// TIA Portal project "13_Buffer_Station" (V19)

(* hardware
DEVICE "S7-1500/ET200MP station_1"  S7-1500 station
   slot 0: "Rail_0"  Rack  6ES7 590-1***0-0AA0
   slot 1: "PLC_1"  CPU 1513-1 PN  6ES7 513-1AL02-0AB0  V2.9
      slot 3: "CPU display_1"  6ES7591-1AA00-0AA0
      slot 32768: "PROFINET interface_1"  X1
         slot 32769: "Port_1"  X1 P1
         slot 32770: "Port_2"  X1 P2
      slot 34817: "Virtual CP interface port_1"  Virtual CP interface port  Virtual CP interface port
*)

// ===== PLC "PLC_1"  CPU 1513-1 PN =====

VAR_GLOBAL   // PLC tag table "Default tag table"
   "nw2" AT %M0.0 : Bool;
   "nw3 2nd memory (Pause)" AT %M0.2 : Bool;
   "nw3 1st memory (Unpause)" AT %M0.1 : Bool;
   "nw3 return" AT %M4.0 : Bool;
   "nw4" AT %M0.3 : Bool;
   "nw6 ae p" AT %M1.3 : Bool;
   "nw6 1st SR" AT %M0.5 : Bool;
   "nw6 abe p" AT %M0.7 : Bool;
   "nw6 abe p2" AT %M1.4 : Bool;
   "nw6 2nd SR" AT %M1.5 : Bool;
   "nw6 ae p2" AT %M1.6 : Bool;
   "nw5" AT %M0.4 : Bool;
   "nw7 1st SR" AT %M0.6 : Bool;
   "I/P for exit conveyor" AT %MD100 : Real;
   "nw7 2nd SR" AT %M1.7 : Bool;
   "nw8 abe p" AT %M1.1 : Bool;
   "nw8" AT %M1.0 : Bool;
   "nw8 ae p" AT %M1.2 : Bool;
   "nw8 ret" AT %M2.0 : Bool;
   "Convert potention meter value from Real to DINT" AT %MD110 : Real;
   "Store MD110 here & send to QD42" AT %MD10 : DInt;
   "nw9 ae p1" AT %M2.2 : Bool;
   "nw9 1st SR" AT %M2.1 : Bool;
   "nw9 abe p1" AT %M2.3 : Bool;
   "nw9 abe p2" AT %M2.4 : Bool;
   "nw9 ae p2" AT %M2.5 : Bool;
   "nw9 abe p3" AT %M2.7 : Bool;
   "nw9 2nd SR" AT %M2.6 : Bool;
   "nw9 ae p3" AT %M3.0 : Bool;
   "nw10 1st SR" AT %M3.1 : Bool;
   "I/P for exit conveyor (set)" AT %MD120 : Real;
   "nw10 2nd SR" AT %M3.2 : Bool;
   "nw11 abe p1" AT %M3.4 : Bool;
   "nw11" AT %M3.3 : Bool;
   "nw11 ae p1" AT %M3.6 : Bool;
   "nw11 ae p2" AT %M3.5 : Bool;
   "nw11 abe p2" AT %M3.7 : Bool;
END_VAR

VAR_GLOBAL   // PLC tag table "Tag table from XML_1"
   "Start" AT %I0.0 : Bool;
   "Pause & Unpause" AT %I0.1 : Bool;
   "Reset" AT %I0.2 : Bool;
   "At buffer entry" AT %I0.3 : Bool;
   "At buffer exit" AT %I0.4 : Bool;
   "At exit" AT %I0.5 : Bool;
   "Without set (mode)" AT %I0.6 : Bool;
   "Send set (mode)" AT %I0.7 : Bool;
   "Start light" AT %Q0.0 : Bool;
   "P & UP light" AT %Q0.1 : Bool;
   "Reset light" AT %Q0.2 : Bool;
   "Stop blade" AT %Q0.3 : Bool;
   "Buffer Vel." AT %ID30 : Real;
   "Set the value for boxes" AT %ID34 : Real;
   "Buffer conveyor" AT %QD30 : Real;
   "Exit conveyor" AT %QD34 : Real;
   "Display Buffer (Speed)" AT %QD38 : Real;
   "Display for set of boxes" AT %QD42 : DInt;
   "Display Counter" AT %QD46 : DInt;
END_VAR

// folder: System blocks/Program resources

DATA_BLOCK "IEC_Counter_0_DB"   // DB1
{ S7_Optimized_Access := 'TRUE' }
AUTHOR : Simatic
FAMILY : IEC
NAME : CNTR
VERSION : 1.0
// stored: InstanceOfName IEC_COUNTER
"IEC_COUNTER"
BEGIN
END_DATA_BLOCK

DATA_BLOCK "IEC_Counter_0_DB_1"   // DB2
{ S7_Optimized_Access := 'TRUE' }
AUTHOR : SIMATIC
FAMILY : IEC
NAME : DCNTR
VERSION : 1.2
// stored: InstanceOfName IEC_DCOUNTER
"IEC_DCOUNTER"
BEGIN
END_DATA_BLOCK

DATA_BLOCK "IEC_Counter_0_DB_2"   // DB3
{ S7_Optimized_Access := 'TRUE' }
AUTHOR : SIMATIC
FAMILY : IEC
NAME : DCNTR
VERSION : 1.2
// stored: InstanceOfName IEC_DCOUNTER
"IEC_DCOUNTER"
BEGIN
END_DATA_BLOCK

DATA_BLOCK "IEC_Counter_0_DB_3"   // DB4
{ S7_Optimized_Access := 'TRUE' }
AUTHOR : SIMATIC
FAMILY : IEC
NAME : DCNTR
VERSION : 1.2
// stored: InstanceOfName IEC_DCOUNTER
"IEC_DCOUNTER"
BEGIN
END_DATA_BLOCK

DATA_BLOCK "IEC_Counter_0_DB_4"   // DB5
{ S7_Optimized_Access := 'TRUE' }
AUTHOR : SIMATIC
FAMILY : IEC
NAME : DCNTR
VERSION : 1.2
// stored: InstanceOfName IEC_DCOUNTER
"IEC_DCOUNTER"
BEGIN
END_DATA_BLOCK

// folder: (top level)

ORGANIZATION_BLOCK "Main"   // OB1, LAD, ProgramCycle
TITLE = "Main Program Sweep (Cycle)"
{ S7_Optimized_Access := 'TRUE' }
VERSION : 0.1
   VAR_INPUT
      Initial_Call : Bool;   // Initial call of this OB
      Remanence : Bool;   // =True, if remanent data are available
   END_VAR
   VAR_TEMP   // added for the SCL form of the ladder/FBD networks
      _w1 : Bool;
      _w2 : Bool;
      _w3 : Bool;
      _w4 : Bool;
      _w5 : Bool;
      _w6 : Bool;
   END_VAR
BEGIN

REGION Network 2: Start or Reset System with LED ON/OFF
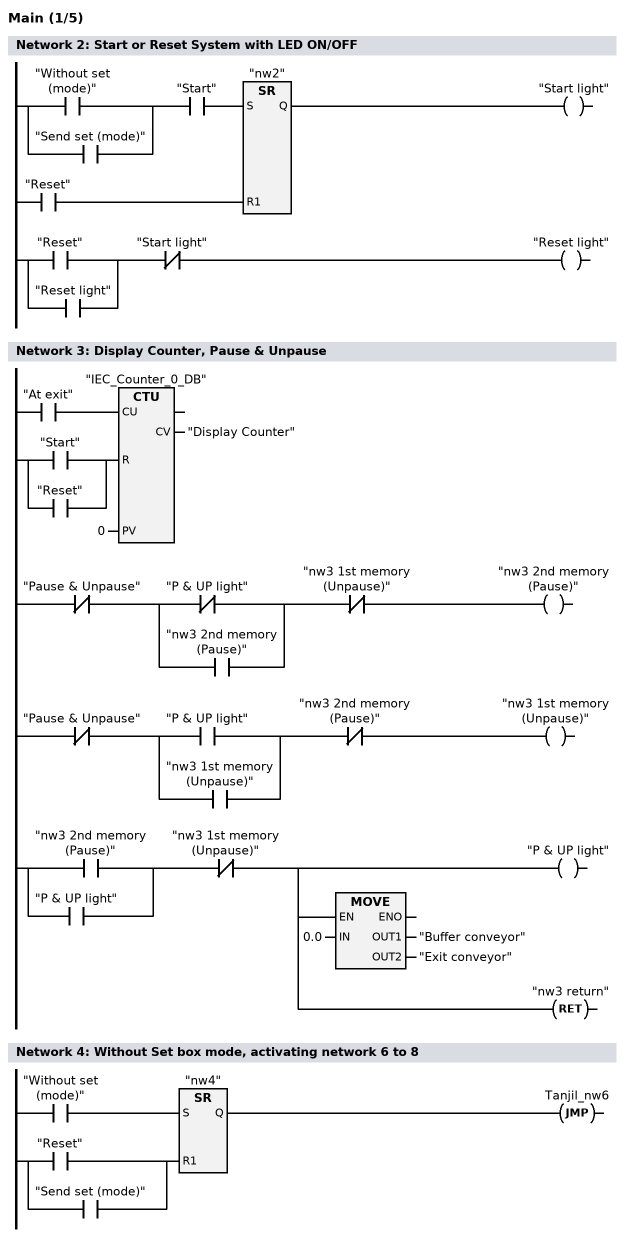
   RUNG wire#powerrail
      Contact( "Without set (mode)" )
      wire#w1
      Contact( "Start" )
      S_SR(operand := "nw2", r1 := wire#w2)
      Coil( "Start light" )
   END_RUNG
   RUNG wire#powerrail
      Contact( "Send set (mode)" )
   END_RUNG wire#w1
   RUNG wire#powerrail
      Contact( "Reset" )
   END_RUNG wire#w2
   RUNG wire#powerrail
      Contact( "Reset" )
      wire#w3
      I_Contact( "Start light" )
      Coil( "Reset light" )
   END_RUNG
   RUNG wire#powerrail
      Contact( "Reset light" )
   END_RUNG wire#w3
   // the same network as SCL:
   IF ("Without set (mode)" OR "Send set (mode)") AND "Start" THEN
       "nw2" := TRUE;   // SR flip-flop
   END_IF;
   IF "Reset" THEN "nw2" := FALSE; END_IF;
   "Start light" := "nw2";
   "Reset light" := ("Reset" OR "Reset light") AND NOT "Start light";
END_REGION

REGION Network 3: Display Counter, Pause & Unpause
   "IEC_Counter_0_DB".CTU(CU := "At exit", R := "Start" OR "Reset", PV := 0, CV => "Display Counter");
   "nw3 2nd memory (Pause)" := NOT "Pause & Unpause" AND (NOT "P & UP light" OR "nw3 2nd memory (Pause)") AND NOT "nw3 1st memory (Unpause)";
   "nw3 1st memory (Unpause)" := NOT "Pause & Unpause" AND ("P & UP light" OR "nw3 1st memory (Unpause)") AND NOT "nw3 2nd memory (Pause)";
   "P & UP light" := ("nw3 2nd memory (Pause)" OR "P & UP light") AND NOT "nw3 1st memory (Unpause)";
   IF "P & UP light" THEN
       "Buffer conveyor" := 0.0;
       "Exit conveyor" := 0.0;
       ENO := "nw3 return";
       RETURN;
   END_IF;
END_REGION

REGION Network 4: Without Set box mode, activating network 6 to 8
   RUNG wire#powerrail
      Contact( "Without set (mode)" )
      S_SR(operand := "nw4", r1 := wire#w1)
      JumpCoil( Tanjil_nw6 )
   END_RUNG
   RUNG wire#powerrail
      Contact( "Reset" )
   END_RUNG wire#w1
   RUNG wire#powerrail
      Contact( "Send set (mode)" )
   END_RUNG wire#w1
   // the same network as SCL:
   IF "Without set (mode)" THEN
       "nw4" := TRUE;   // SR flip-flop
   END_IF;
   IF "Reset" OR "Send set (mode)" THEN "nw4" := FALSE; END_IF;
   IF "nw4" THEN GOTO Tanjil_nw6; END_IF;
END_REGION

REGION Network 5: Activating Network 9 to 11 (sending set of boxes)
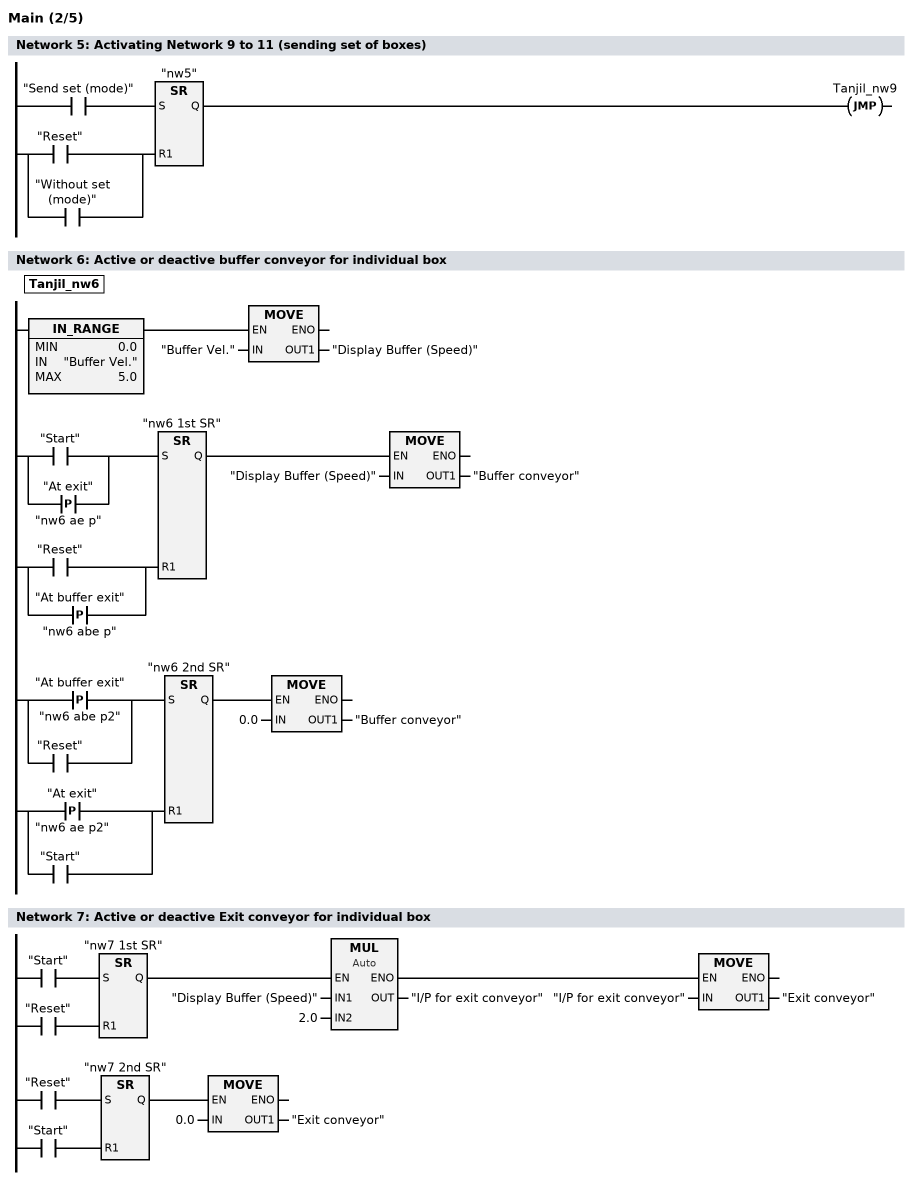
   RUNG wire#powerrail
      Contact( "Send set (mode)" )
      S_SR(operand := "nw5", r1 := wire#w1)
      JumpCoil( Tanjil_nw9 )
   END_RUNG
   RUNG wire#powerrail
      Contact( "Reset" )
   END_RUNG wire#w1
   RUNG wire#powerrail
      Contact( "Without set (mode)" )
   END_RUNG wire#w1
   // the same network as SCL:
   IF "Send set (mode)" THEN
       "nw5" := TRUE;   // SR flip-flop
   END_IF;
   IF "Reset" OR "Without set (mode)" THEN "nw5" := FALSE; END_IF;
   IF "nw5" THEN GOTO Tanjil_nw9; END_IF;
END_REGION

REGION Network 6: Active or deactive buffer conveyor for individual box
   Label( Tanjil_nw6 )
   RUNG wire#powerrail
      { S7_Templates := "SrcType := Real" } InRange(min := 0.0, in := "Buffer Vel.", max := 5.0)
      { S7_GenerateENO := "TRUE" } Move(in := "Buffer Vel.", out1 => "Display Buffer (Speed)")
   END_RUNG
   RUNG wire#powerrail
      Contact( "Start" )
      wire#w1
      S_SR(operand := "nw6 1st SR", r1 := wire#w2)
      { S7_GenerateENO := "TRUE" } Move(in := "Display Buffer (Speed)", out1 => "Buffer conveyor")
   END_RUNG
   RUNG wire#powerrail
      P_Contact(operand := "At exit", bit := "nw6 ae p")
   END_RUNG wire#w1
   RUNG wire#powerrail
      Contact( "Reset" )
   END_RUNG wire#w2
   RUNG wire#powerrail
      P_Contact(operand := "At buffer exit", bit := "nw6 abe p")
   END_RUNG wire#w2
   RUNG wire#powerrail
      P_Contact(operand := "At buffer exit", bit := "nw6 abe p2")
      wire#w3
      S_SR(operand := "nw6 2nd SR", r1 := wire#w4)
      { S7_GenerateENO := "TRUE" } Move(in := 0.0, out1 => "Buffer conveyor")
   END_RUNG
   RUNG wire#powerrail
      Contact( "Reset" )
   END_RUNG wire#w3
   RUNG wire#powerrail
      P_Contact(operand := "At exit", bit := "nw6 ae p2")
   END_RUNG wire#w4
   RUNG wire#powerrail
      Contact( "Start" )
   END_RUNG wire#w4
   // the same network as SCL:
   Tanjil_nw6:
   IF (0.0 <= "Buffer Vel.") AND ("Buffer Vel." <= 5.0) THEN
       "Display Buffer (Speed)" := "Buffer Vel.";
   END_IF;
   #_w1 := "At exit" AND NOT "nw6 ae p";   // rising edge of "At exit"
   "nw6 ae p" := "At exit";
   #_w2 := "At buffer exit" AND NOT "nw6 abe p";   // rising edge of "At buffer exit"
   "nw6 abe p" := "At buffer exit";
   IF "Start" OR #_w1 THEN
       "nw6 1st SR" := TRUE;   // SR flip-flop
   END_IF;
   IF "Reset" OR #_w2 THEN "nw6 1st SR" := FALSE; END_IF;
   IF "nw6 1st SR" THEN "Buffer conveyor" := "Display Buffer (Speed)"; END_IF;
   #_w3 := "At buffer exit" AND NOT "nw6 abe p2";   // rising edge of "At buffer exit"
   "nw6 abe p2" := "At buffer exit";
   #_w4 := "At exit" AND NOT "nw6 ae p2";   // rising edge of "At exit"
   "nw6 ae p2" := "At exit";
   IF #_w3 OR "Reset" THEN
       "nw6 2nd SR" := TRUE;   // SR flip-flop
   END_IF;
   IF #_w4 OR "Start" THEN "nw6 2nd SR" := FALSE; END_IF;
   IF "nw6 2nd SR" THEN "Buffer conveyor" := 0.0; END_IF;
END_REGION

REGION Network 7: Active or deactive Exit conveyor for individual box
   RUNG wire#powerrail
      Contact( "Start" )
      S_SR(operand := "nw7 1st SR", r1 := wire#w1)
      { S7_GenerateENO := "TRUE" } Mul(in1 := "Display Buffer (Speed)", in2 := 2.0, out => "I/P for exit conveyor")
      { S7_GenerateENO := "TRUE" } Move(in := "I/P for exit conveyor", out1 => "Exit conveyor")
   END_RUNG
   RUNG wire#powerrail
      Contact( "Reset" )
   END_RUNG wire#w1
   RUNG wire#powerrail
      Contact( "Reset" )
      S_SR(operand := "nw7 2nd SR", r1 := wire#w2)
      { S7_GenerateENO := "TRUE" } Move(in := 0.0, out1 => "Exit conveyor")
   END_RUNG
   RUNG wire#powerrail
      Contact( "Start" )
   END_RUNG wire#w2
   // the same network as SCL:
   // ENO of a box is taken as its EN; it also drops when the box reports an error
   IF "Start" THEN
       "nw7 1st SR" := TRUE;   // SR flip-flop
   END_IF;
   IF "Reset" THEN "nw7 1st SR" := FALSE; END_IF;
   IF "nw7 1st SR" THEN
       "I/P for exit conveyor" := "Display Buffer (Speed)" * 2.0;
       "Exit conveyor" := "I/P for exit conveyor";
   END_IF;
   IF "Reset" THEN
       "nw7 2nd SR" := TRUE;   // SR flip-flop
   END_IF;
   IF "Start" THEN "nw7 2nd SR" := FALSE; END_IF;
   IF "nw7 2nd SR" THEN "Exit conveyor" := 0.0; END_IF;
END_REGION

REGION Network 8: Active or deactive the STOP Blade
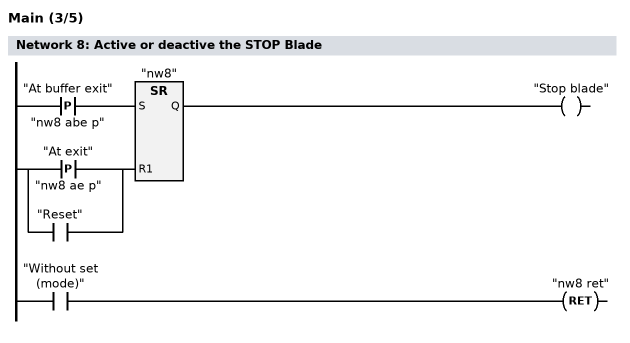
   #_w1 := "At buffer exit" AND NOT "nw8 abe p";   // rising edge of "At buffer exit"
   "nw8 abe p" := "At buffer exit";
   #_w2 := "At exit" AND NOT "nw8 ae p";   // rising edge of "At exit"
   "nw8 ae p" := "At exit";
   IF #_w1 THEN
       "nw8" := TRUE;   // SR flip-flop
   END_IF;
   IF #_w2 OR "Reset" THEN "nw8" := FALSE; END_IF;
   "Stop blade" := "nw8";
   IF "Without set (mode)" THEN
       ENO := "nw8 ret";
       RETURN;
   END_IF;
END_REGION

REGION Network 9: Active Buffer Conveyor
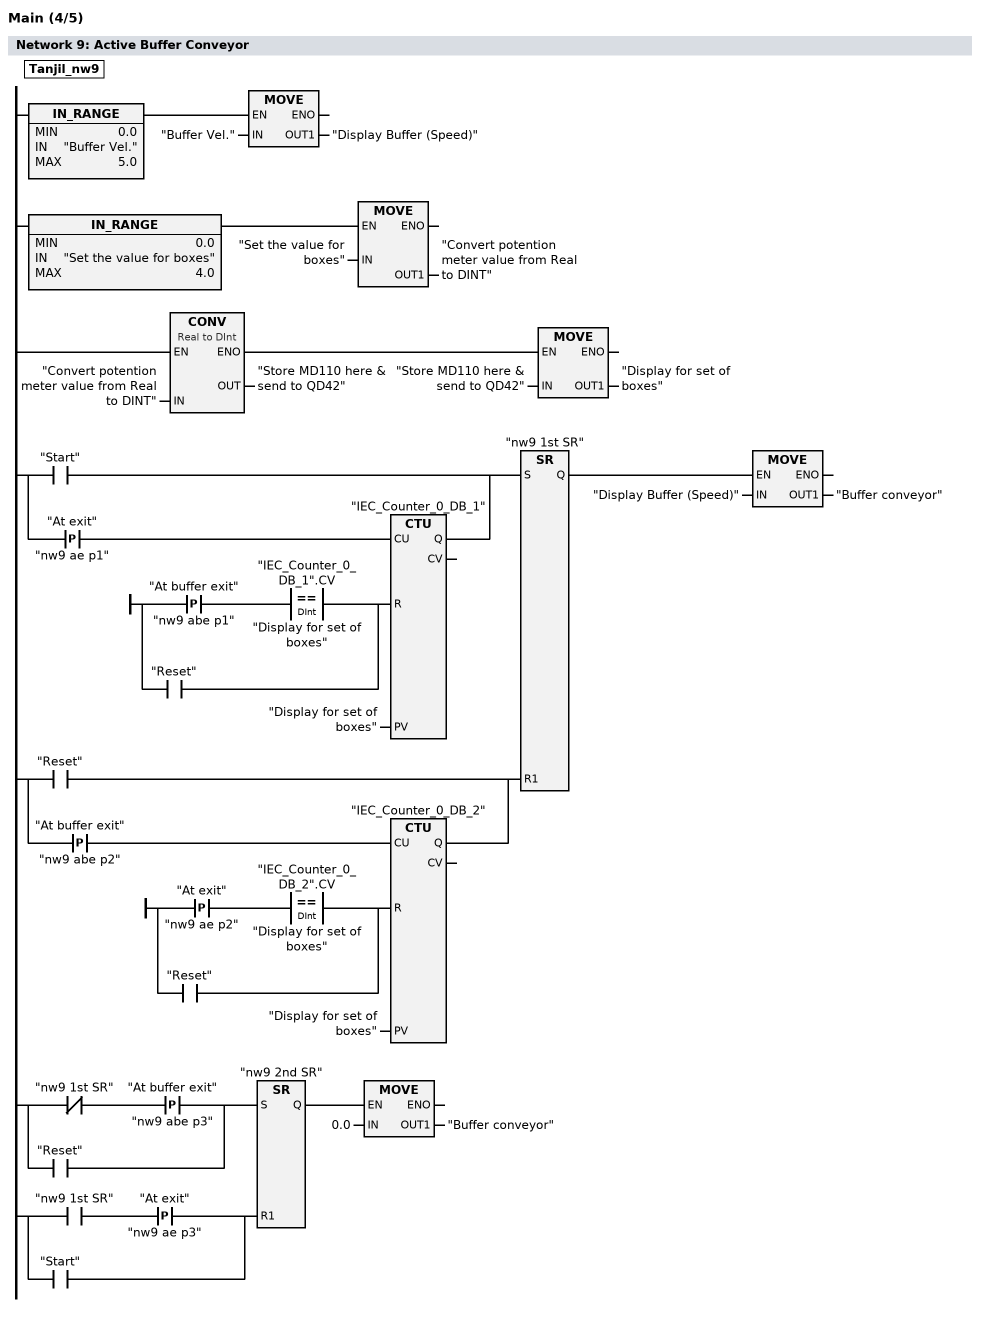
   // ENO of a box is taken as its EN; it also drops when the box reports an error
   Tanjil_nw9:
   IF (0.0 <= "Buffer Vel.") AND ("Buffer Vel." <= 5.0) THEN
       "Display Buffer (Speed)" := "Buffer Vel.";
   END_IF;
   IF (0.0 <= "Set the value for boxes") AND ("Set the value for boxes" <= 4.0) THEN
       "Convert potention meter value from Real to DINT" := "Set the value for boxes";
   END_IF;
   "Store MD110 here & send to QD42" := REAL_TO_DINT("Convert potention meter value from Real to DINT");
   "Display for set of boxes" := "Store MD110 here & send to QD42";
   #_w1 := "At exit" AND NOT "nw9 ae p1";   // rising edge of "At exit"
   "nw9 ae p1" := "At exit";
   #_w2 := "At buffer exit" AND NOT "nw9 abe p1";   // rising edge of "At buffer exit"
   "nw9 abe p1" := "At buffer exit";
   "IEC_Counter_0_DB_1".CTU(CU := #_w1,
                           R := (#_w2 AND ("IEC_Counter_0_DB_1".CV = "Display for set of boxes")) OR "Reset",
                           PV := "Display for set of boxes");
   #_w3 := "At buffer exit" AND NOT "nw9 abe p2";   // rising edge of "At buffer exit"
   "nw9 abe p2" := "At buffer exit";
   #_w4 := "At exit" AND NOT "nw9 ae p2";   // rising edge of "At exit"
   "nw9 ae p2" := "At exit";
   "IEC_Counter_0_DB_2".CTU(CU := #_w3,
                           R := (#_w4 AND ("IEC_Counter_0_DB_2".CV = "Display for set of boxes")) OR "Reset",
                           PV := "Display for set of boxes");
   IF "Start" OR "IEC_Counter_0_DB_1".Q THEN
       "nw9 1st SR" := TRUE;   // SR flip-flop
   END_IF;
   IF "Reset" OR "IEC_Counter_0_DB_2".Q THEN "nw9 1st SR" := FALSE; END_IF;
   IF "nw9 1st SR" THEN "Buffer conveyor" := "Display Buffer (Speed)"; END_IF;
   #_w5 := NOT "nw9 1st SR" AND "At buffer exit" AND NOT "nw9 abe p3";   // rising edge of "At buffer exit"
   "nw9 abe p3" := "At buffer exit";
   #_w6 := "nw9 1st SR" AND "At exit" AND NOT "nw9 ae p3";   // rising edge of "At exit"
   "nw9 ae p3" := "At exit";
   IF #_w5 OR "Reset" THEN
       "nw9 2nd SR" := TRUE;   // SR flip-flop
   END_IF;
   IF #_w6 OR "Start" THEN "nw9 2nd SR" := FALSE; END_IF;
   IF "nw9 2nd SR" THEN "Buffer conveyor" := 0.0; END_IF;
END_REGION

REGION Network 10: Active or deactive EXIT Conveyor
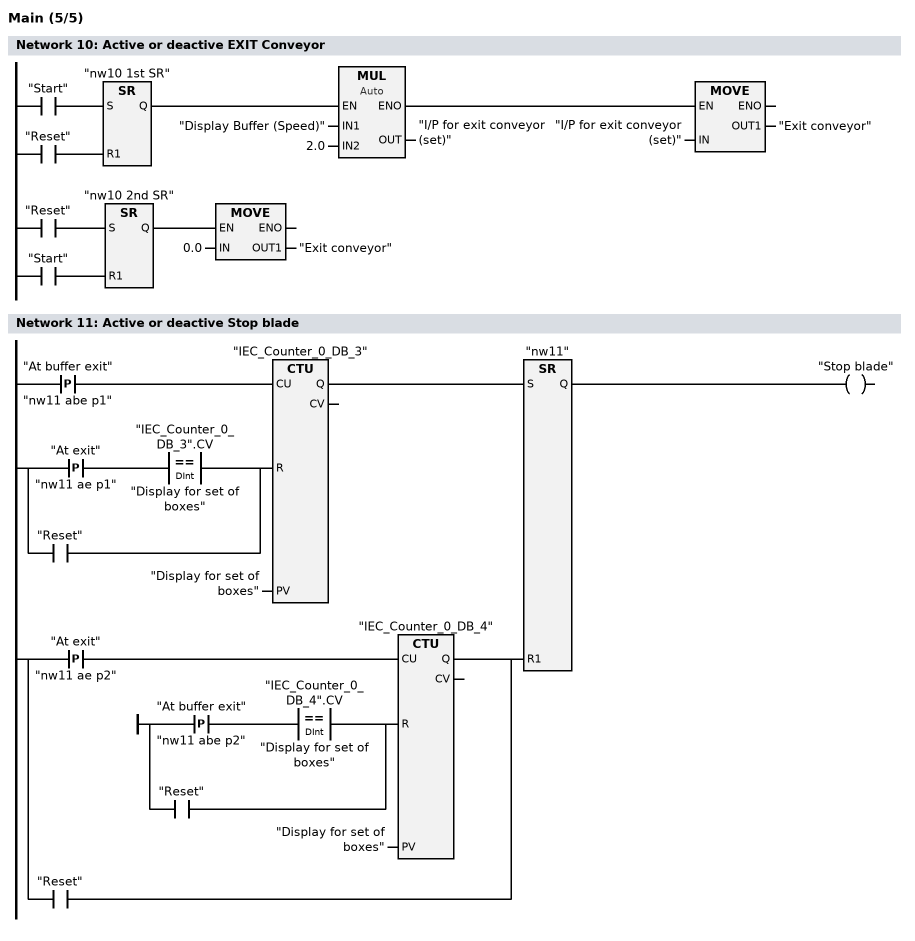
   RUNG wire#powerrail
      Contact( "Start" )
      S_SR(operand := "nw10 1st SR", r1 := wire#w1)
      { S7_GenerateENO := "TRUE" } Mul(in1 := "Display Buffer (Speed)", in2 := 2.0, out => "I/P for exit conveyor (set)")
      { S7_GenerateENO := "TRUE" } Move(in := "I/P for exit conveyor (set)", out1 => "Exit conveyor")
   END_RUNG
   RUNG wire#powerrail
      Contact( "Reset" )
   END_RUNG wire#w1
   RUNG wire#powerrail
      Contact( "Reset" )
      S_SR(operand := "nw10 2nd SR", r1 := wire#w2)
      { S7_GenerateENO := "TRUE" } Move(in := 0.0, out1 => "Exit conveyor")
   END_RUNG
   RUNG wire#powerrail
      Contact( "Start" )
   END_RUNG wire#w2
   // the same network as SCL:
   // ENO of a box is taken as its EN; it also drops when the box reports an error
   IF "Start" THEN
       "nw10 1st SR" := TRUE;   // SR flip-flop
   END_IF;
   IF "Reset" THEN "nw10 1st SR" := FALSE; END_IF;
   IF "nw10 1st SR" THEN
       "I/P for exit conveyor (set)" := "Display Buffer (Speed)" * 2.0;
       "Exit conveyor" := "I/P for exit conveyor (set)";
   END_IF;
   IF "Reset" THEN
       "nw10 2nd SR" := TRUE;   // SR flip-flop
   END_IF;
   IF "Start" THEN "nw10 2nd SR" := FALSE; END_IF;
   IF "nw10 2nd SR" THEN "Exit conveyor" := 0.0; END_IF;
END_REGION

REGION Network 11: Active or deactive Stop blade
   #_w1 := "At buffer exit" AND NOT "nw11 abe p1";   // rising edge of "At buffer exit"
   "nw11 abe p1" := "At buffer exit";
   #_w2 := "At exit" AND NOT "nw11 ae p1";   // rising edge of "At exit"
   "nw11 ae p1" := "At exit";
   "IEC_Counter_0_DB_3".CTU(CU := #_w1,
                           R := (#_w2 AND ("IEC_Counter_0_DB_3".CV = "Display for set of boxes")) OR "Reset",
                           PV := "Display for set of boxes");
   #_w3 := "At exit" AND NOT "nw11 ae p2";   // rising edge of "At exit"
   "nw11 ae p2" := "At exit";
   #_w4 := "At buffer exit" AND NOT "nw11 abe p2";   // rising edge of "At buffer exit"
   "nw11 abe p2" := "At buffer exit";
   "IEC_Counter_0_DB_4".CTU(CU := #_w3,
                           R := (#_w4 AND ("IEC_Counter_0_DB_4".CV = "Display for set of boxes")) OR "Reset",
                           PV := "Display for set of boxes");
   IF "IEC_Counter_0_DB_3".Q THEN
       "nw11" := TRUE;   // SR flip-flop
   END_IF;
   IF "IEC_Counter_0_DB_4".Q OR "Reset" THEN "nw11" := FALSE; END_IF;
   "Stop blade" := "nw11";
END_REGION
END_ORGANIZATION_BLOCK